// TwinCAT 3 PLC project EtherCAT_Test_1
// ProgramVersion: 3.1.4023.0
// libraries:
//   Tc2_EtherCAT, * (Beckhoff Automation GmbH)
//   Tc2_HVAC, * (Beckhoff Automation GmbH)
//   Tc2_Standard, * (Beckhoff Automation GmbH)
//   Tc2_System, * (Beckhoff Automation GmbH)
//   Tc3_Module, * (Beckhoff Automation GmbH)
// project tree:
//   DUTs/ ST_TypeOfPositioning.TcDUT
//   GVLs/ GVL.TcGVL
//   / PlcTask.TcTTO
//   POUs/ MAIN.TcPOU, P_ProfilePositionModeTest.TcPOU, StartUpTests.TcPOU, ST_PlcErrorStartUp.TcDUT
//   POUs/ProfilePositionMode/ FB_EnableDevice.TcPOU, Motion.TcPOU
// real-time tasks:
//   TASK PlcTask: cycle T#10ms, priority 20, ADS port 350
// motion (NC):
//   TASK NC-Task 1 SAF: cycle T#2ms, priority 4, ADS port 501
//   TASK NC-Task 1 SVB: cycle T#10ms, priority 8, ADS port 511
//   AXIS Axis 1 (id 1)
//     OtherSettings: AllowMotionCmdToSlave=true
//     encoder EncType=19
//       EncPara: MaxCount=#xffffffff
//     drive DrvType=16
//       DrvPara: MaxCount=#xffffffff
//         Analog: TorqueSetpointScale=10, ScaleFactorActTorque=0.1
//         TimeComp: TaskDelayCycles=1
//     controller CtrType=1
//       CtrPara: PriorControlFactor=1
//         Observer: BandWidth=20
// I/O:
//   DEVICE Device 1 (EtherCAT), AmsNetId 5.109.65.175.2.1
//     Term 1 (EK1200) [EK1200-5000 EtherCAT Power supply (2A E-Bus)]
//       Term 2 (EL1859) [EL1859 8Ch. Dig. Input 24V, 3ms, 8Ch. Dig. Output 24V, 0.5A]
//       Term 3 (EL6751) [EL6751 CANopen Master]
//       Term 4 (EK1110) [EK1110 EtherCAT extension]
//     Drive 5 (HTB) [HTB]
//       modules: Module 1 (csp - axis)

CONFIGURATION EtherCAT_Test_1
    RESOURCE PLC ON TwinCAT3
        TASK PlcTask(INTERVAL := T#10ms, PRIORITY := 20);
        PROGRAM MAIN WITH PlcTask : MAIN;
    END_RESOURCE
END_CONFIGURATION

// ---- DUTs/ST_TypeOfPositioning.TcDUT
TYPE ST_TypeOfPositioning :
STRUCT
	bStartImmediately			: BOOL; (*if Bool is true, target position is absolute, otherwise relative*)
	bAbsolutePositioning		: BOOL; (*if Bool is true, velocity does not change, when first target position is reached - no braking*)
	bChangeOnSetPoint			: BOOL; (*if set true, moving command is executed immediately*)
	nReferencing				: BYTE;
	(*describes positioning behaviour 
		- 1: Positioning relative to previous target position
		- 2: Positioning relative to default value of ramp generator
		- 3: Positioning relative to actual position*)	
END_STRUCT
END_TYPE

// ---- POUs/ST_PlcErrorStartUp.TcDUT
TYPE ST_PlcErrorStartUp :
STRUCT
	bPlcError		: BOOL;
	bErrorCode		: ARRAY[1..4] OF UDINT;
END_STRUCT
END_TYPE

// ---- GVLs/GVL.TcGVL
{attribute 'qualified_only'}
VAR_GLOBAL
	sNetId				: T_AmsNetId := '5.109.65.175.2.1';
	nSlaveAddr			: UINT := 1004;
	
	Controlword AT%Q*		: UINT;	
	Statusword AT%I*		: UINT;
END_VAR

// ---- POUs/MAIN.TcPOU
PROGRAM MAIN
VAR_INPUT
	Controlword AT%Q*		: UINT;	
	TargetPosition AT%Q*	: DINT;
END_VAR
VAR_OUTPUT
	Statusword AT%I*		: UINT;
END_VAR
VAR
	bStartUpTest			: BOOL;
END_VAR	

VAR
	aTemperatureObjects		: ARRAY[1..2] OF INT := [1,1]; 	//0x2200, 0x2202
	aMOPObjects				: ARRAY[1..2] OF INT := [1,1]; 	//0x6060, 0x6061
	aControlStatusWords		: ARRAY[1..2] OF INT := [1,1]; 	//0x6040, 0x6041
	bTargetPosition			: BOOL;							//0x607A
	
	fbSetToPPMode			: FB_EcCoeSdoWrite;
	bSetToPPMode			: BOOL;
	tSetToPPMode			: TON;
	nModeOfOperation		: UDINT := 1;
END_VAR

//StartUpTests(bTrigger := bStartUpTest,
//	aTemperatureObjects := aTemperatureObjects,
//	aControlStatusWords := aControlStatusWords,
//	aMOPObjects := aMOPObjects,
//	sNetID := GVL.sNetId,
//	nSlaveAddr := GVL.nSlaveAddr);

fbSetToPPMode(sNetId := GVL.sNetId, 
				nSlaveAddr := GVL.nSlaveAddr,
				nIndex := 16#6060,
				pSrcBuf := ADR(nModeOfOperation),
				cbBufLen := SIZEOF (nModeOfOperation),
				bExecute := bSetToPPMode);
tSetToPPMode(IN := bSetToPPMode,
				PT := T#250MS);
bSetToPPMode := TRUE;
IF tSetToPPMode.Q THEN
	P_ProfilePositionModeTest();	
END_IF

				



//Hallo Julian

END_PROGRAM

// ---- POUs/P_ProfilePositionModeTest.TcPOU
PROGRAM P_ProfilePositionModeTest
VAR
	fbMoveInProfilePosition			: Motion;
	fbGetCurrentPosition			: FB_EcCoeSdoRead;
	fbGetStatusword					: FB_EcCoeSdoRead;
	fbGetPositionWindow				: FB_EcCoeSdoRead;
	fbGetPositionDemandValue		: FB_EcCoeSdoRead;
	tWaitForCurrentPosition			: TON;
	tWaitForPositionDemandValue		: TON;
	tGetStatusword					: TON;
	bGetCurrentPosition				: BOOL;
	bMove							: BOOL; 
	bExecuteTimer					: BOOL;
	bGetStatusword					: BOOL;
	bGetParameters					: BOOL;
	bSetPositioningOptionCode		: BOOL;
	bGetPositionDemandValue			: BOOL;
	bBasicOperationAbsStarted		: BOOL;
	bBasicOperationAbsFinished		: BOOL := FALSE;
	bPositioningOptionCodeSet		: BOOL;
	bTargetReached					: BOOL;
	bTestAbsolutePositioning		: BOOL;
	nTargetPosition					: DINT;
	nCurrentPosition				: DINT;
	nTargetPositionBuf				: DINT;
	nPositionDemandValue			: DINT;
	nStatusword						: UINT;
	nPositionWindow					: UDINT;
	
	
	bTest							: BOOL;
	bAusprobieren					: BOOL;
END_VAR

VAR
	bBasicOperationAbs				: BOOL;
	bBasicOperationRel				: BOOL;
	bPositioningOptionCode			: BOOL;
END_VAR

//For Test Set of Setpoints
VAR
	bSetOfSetpointFinished 			: BOOL;
	nCurrentPositionBuf				: DINT;
	bSetPointSet					: BOOL;  //For both
	bSetOfSetpoints					: BOOL;
	bStartBasicOperationAbs			: BOOL;
	bTestSetOfSetpoints				: BOOL;
	bSetOfSetpointsFinished			: BOOL;
END_VAR

//Fo Test Change Immediately
VAR
	bTestChangeImmediately			: BOOL;
	bChangeImmediatelyFinished		: BOOL;
	bChangeImmediately				: BOOL;
END_VAR

//For test of relative Positioninig
VAR
	tSetPositioningOptionCode		: TON;
	fbSetPositioningOptionCode		: FB_EcCoeSdoWrite;
	bTestRelativePositioning		: BOOL;
	bRelativePositioningFinished	: BOOL;
	nPositioningOptionCode			: DINT;
	nCounter						: DINT;
END_VAR

tWaitForCurrentPosition(IN := bGetCurrentPosition,
							PT := T#10MS);
tGetStatusword(IN := bGetStatusword,
					PT := T#500MS);	
tSetPositioningOptionCode(IN := bSetPositioningOptionCode,
							PT := T#125MS);		
tWaitForPositionDemandValue(IN := bGetPositionDemandValue,
							PT := T#125MS);
IF tWaitForCurrentPosition.Q THEN
	bGetCurrentPosition := FALSE;
ELSE
	bGetCurrentPosition := TRUE;		
END_IF
fbMoveInProfilePosition(sNetID := GVL.sNetId,
						nSlaveAddr := GVL.nSlaveAddr,
						nTargetPosition := nTargetPosition,
						bMove := bMove);
fbGetStatusword(sNetId := GVL.sNetId,
				nSlaveAddr := GVL.nSlaveAddr,
				nIndex := 16#6041,
				nSubindex := 0,
				pDstBuf := ADR(nStatusWord),
				cbBufLen := SIZEOF(nStatusWord),
				bExecute := bGetStatusword);
fbGetCurrentPosition(sNetId := GVL.sNetId,
						nSlaveAddr := GVL.nSlaveAddr,
						nIndex := 16#6064,
						nSubIndex := 0,
						pDstBuf := ADR(nCurrentPosition),
						cbBufLen := SIZEOF(nCurrentPosition),
						bExecute := bGetCurrentPosition);
fbGetPositionWindow(sNetId := GVL.sNetId,
					nSlaveAddr := GVL.nSlaveAddr,
					nIndex := 16#6067,
					nSubIndex := 0,
					pDstBuf := ADR(nPositionWindow),
					cbBufLen := SIZEOF(nPositionWindow),
					bExecute := bGetParameters);
fbGetPositionDemandValue(sNetId := GVL.sNetId,
							nSlaveAddr := GVL.nSlaveAddr,
							nIndex := 16#60FC,
							nSubIndex := 0,
							pDstBuf := ADR(nPositionDemandValue),
							cbBufLen := SIZEOF(nPositionDemandValue),
							bExecute := bGetPositionDemandValue);
fbSetPositioningOptionCode(sNetId := GVL.sNetId,
							nSlaveAddr := GVL.nSlaveAddr,
							nIndex := 16#60F2,
							nSubindex := 0,
							pSrcBuf := ADR(nPositioningOptionCode),
							cbBufLen := SIZEOF(nPositioningOptionCode),
							bExecute := bSetPositioningOptionCode);
bGetParameters := TRUE;

IF bStartBasicOperationAbs THEN					
	//Basic Operation
	//Set-point is applied to the device
	//Move to absolute position is tested
	//Wait until Target reach Bit is set
	//Control if position is within error window
	
	//Target shall be an absolute value
	MAIN.Controlword.6 := 0;

	//Operation has not yet started and we are sure that initial position is obtained
	IF NOT bBasicOperationAbsStarted THEN
		nTargetPosition := nCurrentPosition + 5000000;
		//Start absolute positioning
		bMove := TRUE;	
		bBasicOperationAbsStarted := TRUE;
	END_IF
					
	//Target reached?
	bGetStatusword := TRUE;
	IF tGetStatusword.Q THEN
		IF NOT nStatusword.10 THEN
			bGetStatusword := FALSE;
		ELSIF ((nCurrentPosition >= nTargetPosition - nPositionWindow)
				AND (nCurrentPosition <= nTargetPosition + nPositionWindow)) 
				AND fbMoveInProfilePosition.bStartPositioning THEN
			//absolute Positionining
			bBasicOperationAbs := TRUE;
			bBasicOperationAbsFinished := TRUE;
			bStartBasicOperationAbs := FALSE;
		ELSIF fbMoveInProfilePosition.bStartPositioning THEN
			bBasicOperationAbs := FALSE;
			bBasicOperationAbsFinished := TRUE;
			bStartBasicOperationAbs := FALSE;
		END_IF
		bGetStatusword := FALSE;
	END_IF
END_IF

//Test SetOfSetpoints
IF bTestSetOfSetpoints AND bBasicOperationAbsFinished AND NOT bSetOfSetpointsFinished THEN
	IF NOT bSetPointSet THEN
		MAIN.Controlword.5 := 0;
		nTargetPosition := nCurrentPosition + 100000000;
		nTargetPositionBuf := nTargetPosition;
		nCurrentPositionBuf := nCurrentPosition + 10000000/2;
		bSetPointSet := TRUE;
	END_IF
	IF (nCurrentPosition > nCurrentPositionBuf) AND bSetPointSet THEN
		nTargetPosition := nCurrentPositionBuf - 10000000/2;
	END_IF
	bSetOfSetpoints := TestChangeOfSetpoints(bActive => bSetOfSetpointsFinished);
	IF bSetOfSetpointsFinished THEN
		bSetPointSet := FALSE;
	END_IF
END_IF

//Change Immediately
IF bTestChangeImmediately AND bSetOfSetpointsFinished AND NOT bChangeImmediatelyFinished THEN
	IF NOT bSetPointSet THEN
		MAIN.Controlword.5 := 1;
		nTargetPosition := nCurrentPosition + 100000000;
		nTargetPositionBuf := nTargetPosition;
		nCurrentPositionBuf := nCurrentPosition + 10000000/2;
		bSetPointSet := TRUE;
	END_IF
	IF (nCurrentPosition > nCurrentPositionBuf) AND bSetPointSet THEN
		nTargetPosition := nCurrentPositionBuf - 10000000/2;
	END_IF
	bChangeImmediately := NOT TestChangeOfSetpoints(bActive => bChangeImmediatelyFinished);
END_IF

//Test relative positioning:
//Bit 6 of Controlword is set to 1

IF bTestRelativePositioning THEN
	MAIN.Controlword.6 := 1;
	//positioning option code: 0
	//Positioning moves shall be performed relative to the preciding
	//target position
	IF nCounter = 0 THEN
		nPositioningOptionCode := 0;
		IF tSetPositioningOptionCode.Q THEN
			nTargetPosition := 5000000;
		END_IF
		
		nCounter := nCounter + 1;
	END_IF

	//positioning option code: 2#0001
	//Positioning moves shall be performed relative to the actual
	//positioning demand value (16#60FC)
	
	//positioning option code : 2#0010
	//Positioning moves shall be performed relative to the position
	//actual value (16#6064)
END_IF

//test

METHOD TestChangeOfSetpoints : BOOL
VAR_OUTPUT
	bActive		: BOOL;
END_VAR
IF ((nCurrentPosition >= nTargetPositionBuf - nPositionWindow)
	AND (nCurrentPosition <= nTargetPositionBuf + nPositionWindow)) THEN
	bActive := TRUE;
	bSetOfSetPointsFinished := TRUE;
ELSIF ((nCurrentPosition >= nTargetPosition - nPositionWindow)
	AND (nCurrentPosition <= nTargetPosition + nPositionWindow)) THEN
	TestChangeOfSetpoints := FALSE;
	bActive := TRUE;
END_IF
END_METHOD

END_PROGRAM

// ---- POUs/ProfilePositionMode/Motion.TcPOU
FUNCTION_BLOCK Motion
VAR_INPUT
	sNetID					: T_AmsNetId;
	nSlaveAddr				: UINT;
	nTargetPosition			: DINT;
END_VAR
VAR_OUTPUT
	bSuccess				: BOOL;
	bSetpointSet			: BOOL;
	bStartPositioning		: BOOL;
END_VAR
VAR_IN_OUT
//	aControlStatusWords		: ARRAY[1..2] OF INT; 			//0x6040 (Controlword), 0x6041 (Statusword)  
//	bTargetPosition			: BOOL;							//0x607A (Target Position)
	bMove					: BOOL;
END_VAR
VAR
	eMotionState			: (WAIT_FOR_TRIGGER, ENABLE_DEVICE, SET_SETPOINT, VALIDATE_SETPOINT, ACKNOWLEDGE_SET_POINT, WAIT_FOR_NEW_SETPOINT);
	fbEnableDevice			: FB_EnableDevice;
	fbSetSetpoint			: FB_EcCoeSdoWrite;
	fbGetStatusword			: FB_EcCoeSdoRead;
	tWait					: TON;
	tWait2					: TON;
	rTrig					: R_TRIG;
	nStatusword				: UINT;
	bGetStatusword			: BOOL;
	bExecuteWait			: BOOL;
	bSetSetpoint			: BOOL;
	nSetPointBuf			: DINT;
END_VAR

CASE eMotionState OF
	WAIT_FOR_TRIGGER:
		MAIN.Controlword := 0;
		bStartPositioning := FALSE;
		IF bMove THEN
			bSetpointSet := TRUE;
			bSuccess := TRUE;
			ADSLOGSTR(msgCtrlMask := ADSLOG_MSGTYPE_HINT,
				msgFmtStr := 'Enable Device',
				strArg := '');
			eMotionState := ENABLE_DEVICE;
		END_IF	

	ENABLE_DEVICE:
		fbEnableDevice (bTrigger := bMove,
						bSuccess => bSuccess,
						sNetId := sNetId,
						nSlaveAddr := nSlaveAddr);
		IF fbEnableDevice.bFinished THEN
			IF NOT bSuccess THEN
//				aControlStatusWords[1] := 0;
//				aControlStatusWords[2] := 0;
				ADSLOGSTR(msgCtrlMask := ADSLOG_MSGTYPE_HINT,
					msgFmtStr := 'Device not successfully enabled',
					strArg := '');
				eMotionState := WAIT_FOR_TRIGGER;
			ELSE
				ADSLOGSTR(msgCtrlMask := ADSLOG_MSGTYPE_HINT,
					msgFmtStr := 'Device successfully enabled',
					strArg := '');
				eMotionState := SET_SETPOINT;
			END_IF
		END_IF
		
	WAIT_FOR_NEW_SETPOINT:
		IF nTargetPosition <> nSetPointBuf THEN
			ADSLOGSTR(msgCtrlMask := ADSLOG_MSGTYPE_HINT,
				msgFmtStr := 'Set Setpoint',
				strArg := '');
				bStartPositioning := FALSE;
			eMotionState := SET_SETPOINT;
		END_IF
		
	SET_SETPOINT:
		bSetpointSet	:= TRUE;
		nSetPointBuf := nTargetPosition;
		fbSetSetpoint(sNetId := sNetID,
					nSlaveAddr := nSlaveAddr,
					nSubIndex := 0,
					nIndex := 16#607A,
					pSrcBuf := ADR(nTargetPosition),
					cbBufLen := SIZEOF(nTargetPosition),
					bExecute := bSetSetpoint);
		bSetSetpoint := TRUE;
		MAIN.TargetPosition := nTargetPosition;
		tWait(IN := bExecuteWait,
				PT := T#175MS); 
		bExecuteWait := TRUE;
		IF tWait.Q THEN
			bExecuteWait := FALSE;
			IF fbSetSetpoint.bError THEN
				//Error when setting Target Position
				bSuccess := FALSE;
				bSetSetpoint := FALSE;
				eMotionState := WAIT_FOR_TRIGGER;
			ELSE
				ADSLOGSTR(msgCtrlMask := ADSLOG_MSGTYPE_HINT,
					msgFmtStr := 'Validate Setpoint',
					strArg := '');
				eMotionState := VALIDATE_SETPOINT;
			END_IF
		END_IF
 
	VALIDATE_SETPOINT:
		bExecuteWait := TRUE;
		MAIN.Controlword.4 := 1;
		fbGetStatusword(sNetId := sNetId,
			nSlaveAddr := nSlaveAddr,
			nIndex := 16#6041,
			nSubIndex := 0,
			pDstBuf := ADR(nStatusword),
			cbBufLen := SIZEOF(nStatusword),
			bExecute := bGetStatusword);
		IF tWait.Q THEN
			bExecuteWait := FALSE;
			tWait2(IN := bGetStatusword,
				PT := T#250MS);
			bGetStatusword := TRUE;
			IF tWait2.Q THEN
				bGetStatusword := FALSE;
				IF nStatusword.12 THEN
					eMotionState := ACKNOWLEDGE_SET_POINT;
				ELSE 
					bSetSetpoint := FALSE;
					bSuccess := FALSE;
//					aControlStatusWords[1] := 0;
//					aControlStatusWords[2] := 0;
					ADSLOGSTR(msgCtrlMask := ADSLOG_MSGTYPE_HINT,
						msgFmtStr := 'Error when validating setpoint',
						strArg := '');
					eMotionState := WAIT_FOR_TRIGGER;
				END_IF
			END_IF
		END_IF
		
	ACKNOWLEDGE_SET_POINT:
		ADSLOGSTR(msgCtrlMask := ADSLOG_MSGTYPE_HINT,
			msgFmtStr := 'Acknowledge Setpoint',
			strArg := '');
		bGetStatusword := TRUE;
		IF tWait2.Q AND nStatusword.12 THEN
			bStartPositioning := TRUE;
			bGetStatusword := FALSE;
			//Set point acknowledge is set back
			MAIN.Controlword.4 := 0;
			ADSLOGSTR(msgCtrlMask := ADSLOG_MSGTYPE_HINT,
				msgFmtStr := 'Wait for new Setpoint',
				strArg := '');
			eMotionState := WAIT_FOR_NEW_SETPOINT;
		ELSE
			//TODO FAULT
			eMotionState := WAIT_FOR_TRIGGER;
		END_IF
END_CASE

END_FUNCTION_BLOCK

// ---- POUs/ProfilePositionMode/FB_EnableDevice.TcPOU
FUNCTION_BLOCK FB_EnableDevice 
VAR_IN_OUT
	bTrigger			: BOOL;
END_VAR
VAR_INPUT
	sNetID				: T_AmsNetId;
	nSlaveAddr			: UINT;
END_VAR
VAR_OUTPUT
	bFinished			: BOOL;
	bSuccess			: BOOL;
END_VAR
VAR
	eState				: (WAIT_FOR_TRIGGER, SHUTDOWN, SWITCH_ON);
	tWait1				: TON;
	tWait2				: TON;
	fbGetStatusword		: FB_EcCoeSdoRead;
	nStatusword			: UINT;
	bGetStatusword		: BOOL;
	bExecuteTimer		: BOOL;
END_VAR

CASE eState OF
	WAIT_FOR_TRIGGER:
		IF bTrigger THEN
			bExecuteTimer	:= FALSE;
			bSuccess := TRUE;
			bFinished := FALSE;
			bTrigger := FALSE;
			eState := SHUTDOWN;
		END_IF
	
	SHUTDOWN:
		MAIN.Controlword.0 := 0;
		MAIN.Controlword.1 := 1;
		MAIN.Controlword.2 := 1;
		MAIN.Controlword.7 := 0;

		tWait1(PT := T#125MS,
			IN := bExecuteTimer);
			bExecuteTimer := TRUE;
		IF tWait1.Q THEN
			bExecuteTimer := FALSE;
			tWait2(IN := bGetStatusword,
				PT := T#250MS);
			fbGetStatusword(sNetId := sNetId,
				nSlaveAddr := nSlaveAddr,
				nIndex := 16#6041,
				nSubIndex := 0,
				pDstBuf := ADR(nStatusword),
				cbBufLen := SIZEOF(nStatusword),
				bExecute := bGetStatusword);
			bGetStatusword := TRUE;
			IF tWait2.Q THEN
				ADSLOGSTR(msgCtrlMask := ADSLOG_MSGTYPE_HINT,
					msgFmtStr := 'Shutdown',
					strArg := '');
				bExecuteTimer := FALSE;
				IF (nStatusword.0 = 1 AND nStatusword.5) 
					AND NOT (nStatusword.1 AND nStatusword.2 AND nStatusword.3
						AND nStatusword.6) THEN
 					eState := SWITCH_ON;
				ELSE 
					bSuccess := FALSE;
					bFinished := TRUE;
					eState := WAIT_FOR_TRIGGER;
				END_IF
			END_IF
		END_IF
		
	SWITCH_ON:
		ADSLOGSTR(msgCtrlMask := ADSLOG_MSGTYPE_HINT,
			msgFmtStr := 'Switch On',
			strArg := '');
		MAIN.Controlword.0 := 1;
		MAIN.Controlword.1 := 1;
		MAIN.Controlword.2 := 1;
		Main.Controlword.3 := 1;
		Main.Controlword.7 := 0;
		bExecuteTimer := TRUE;
		bGetStatusWord := TRUE;
		IF tWait1.Q THEN
			bExecuteTimer	:= FALSE;
			IF tWait2.Q THEN
				bGetStatusword := FALSE;
				IF nStatusword.0 AND nStatusword.1 AND nStatusword.5 
						AND NOT (nStatusword.2 AND nStatusword.3 AND nStatusword.6) THEN
					bSuccess := FALSE;
				END_IF
				bFinished := TRUE;
				eState := WAIT_FOR_TRIGGER;
			END_IF
		END_IF
END_CASE

END_FUNCTION_BLOCK

// ---- POUs/StartUpTests.TcPOU
PROGRAM StartUpTests
VAR CONSTANT
	stPlcErrorInit			: ST_PlcErrorStartUp := (bPlcError := FALSE, bErrorCode := [0,0,0,0]);
END_VAR

VAR
	eStartUpState 			: (WAIT_FOR_TRIGGER, TEST_SWITCH_ON_DISABLED, 
								SET_MODE_OF_OPERATION, TEST_MODE_OF_OPERATION, GET_TEMPERATURE, CHECK_PLC_ERROR);
	fbSetModeOfOperation	: FB_EcCoeSdoWrite;
	fbGetModeOfOperation	: FB_EcCoeSdoRead;
	fbGetDriveTemperature	: FB_EcCoeSdoRead;
	fbGetMotorTemperature	: FB_EcCoeSdoRead;
	stPlcError				: ST_PlcErrorStartUp;
	tTimeout				: TON;
	tWait1					: TON;
	tWait2					: TON;
	tWait					: TON;
	counter					: INT := -1;
	modeOfOperation			: INT;
	bExecuteChangeMOP		: BOOL;	
	bTestChangeMOP			: BOOL;
END_VAR
VAR_IN_OUT
	bTrigger				: BOOL;
	aTemperatureObjects		: ARRAY[1..2] OF INT;
	aMOPObjects				: ARRAY[1..2] OF INT;
	aControlStatusWords		: ARRAY[1..2] OF INT;
END_VAR
VAR_OUTPUT
	bSwitchOnDisabled		: BOOL;
	bChangeModeOfOperation	: BOOL := TRUE;
	bFinished				: BOOL;
	nDriveTemperature		: INT;
	nMotorTemperature		: INT;
END_VAR
VAR_INPUT
	sNetID					: T_AmsNetId;
	nSlaveAddr				: UINT;
END_VAR

CASE eStartUpState OF
	WAIT_FOR_TRIGGER:
		IF bTrigger THEN
			bTrigger := FALSE;
			tTimeout.IN := FALSE;
			bSwitchOnDisabled := FALSE;
			bChangeModeOfOperation := FALSE;
			bFinished := FALSE;
			counter := 1;
			stPlcError := stPlcErrorInit;
			eStartUpState := TEST_SWITCH_ON_DISABLED;
		END_IF
	
	TEST_SWITCH_ON_DISABLED:
		tTimeout(IN := TRUE,
			PT := T#1000MS);
		IF MAIN.Statusword.6 THEN
			bSwitchOnDisabled := TRUE;
			eStartUpState := SET_MODE_OF_OPERATION;
		ELSIF tTimeout.Q THEN
			bSwitchOnDisabled := FALSE;
			aControlStatusWords[1] := 0;
			eStartUpState := SET_MODE_OF_OPERATION;
		END_IF
	
	SET_MODE_OF_OPERATION:
	bTestChangeMOP := FALSE;
		fbSetModeOfOperation(sNetId := sNetId,
							nSlaveAddr := nSlaveAddr,
							nSubIndex := 0,
							nIndex := 16#6060,
							pSrcBuf := ADR(counter),
							cbBufLen := SIZEOF(counter),
							bExecute := bExecuteChangeMOP);
		tWait1(PT := T#2S, 
			IN := bExecuteChangeMOP);
		bExecuteChangeMOP := TRUE;				
		IF tWait1.Q THEN
			eStartUpState := TEST_MODE_OF_OPERATION;
		END_IF

	TEST_MODE_OF_OPERATION:
		bExecuteChangeMOP := FALSE;	
		fbGetModeOfOperation(sNetId := sNetId,
							nSlaveAddr := nSlaveAddr,
							nSubIndex := 0,
							nIndex := 16#6061,
							pDstBuf := ADR(modeOfOperation),
							cbBufLen := SIZEOF(modeOfOperation),
							bExecute := bTestChangeMOP);
		tWait2(PT := T#2S,
				IN := bTestChangeMOP);
		bTestChangeMOP := TRUE; 
		IF tWait2.Q THEN
			IF NOT modeOfOperation = counter AND counter <> 5 THEN
				bChangeModeOfOperation := FALSE;
				aMOPObjects[1] := 0;
				aMOPObjects[2] := 0;
			END_IF
			counter := counter + 1;
			IF counter < 11 THEN
				eStartUpState := SET_MODE_OF_OPERATION;
			ELSE
				eStartUpState := GET_TEMPERATURE;
			END_IF
		END_IF
	
	GET_TEMPERATURE:
		fbGetDriveTemperature(sNetId := sNetId,
							nSlaveAddr := nSlaveAddr,
							nSubIndex := 0,
							nIndex := 16#2200,
							pDstBuf := ADR(nDriveTemperature),
							cbBufLen := SIZEOF(nDriveTemperature),
							bExecute := TRUE);
		fbGetMotorTemperature(sNetId := sNetId,
							nSlaveAddr := nSlaveAddr,
							nSubIndex := 0,
							nIndex := 16#2202,
							pDstBuf := ADR(nMotorTemperature),
							bExecute := TRUE);							
		tWait(IN := TRUE,
			PT := T#125MS);
		IF tWait.Q THEN
			tWait.IN := FALSE;
		//	eStartUpState := CHECK_PLC_ERROR;
		END_IF
		
		CHECK_PLC_ERROR:
			IF fbSetModeOfOperation.bError OR fbGetModeOfOperation.bError OR
				fbGetDriveTemperature.bError OR fbGetMotorTemperature.bError THEN
				stPlcError.bPlcError := TRUE;
				IF fbSetModeOfOperation.bError THEN
					stPlcError.bErrorCode[1] := fbSetModeOfOperation.nErrId;
					aMOPObjects[1] := 0;
				END_IF
				IF fbGetModeOfOperation.bError THEN
					stPlcError.bErrorCode[2] := fbGetModeOfOperation.nErrId;
					aMOPObjects[2] := 0;		
				END_IF
				IF fbGetDriveTemperature.bError THEN
					stPlcError.bErrorCode[3] := fbGetDriveTemperature.nErrId;
					aTemperatureObjects[1] := 0;
				END_IF
				IF fbGetMotorTemperature.bError THEN
					stPlcError.bErrorCode[4] := fbGetMotorTemperature.nErrId;
					aTemperatureObjects[2] := 0;
				END_IF
			END_IF
			bFinished := TRUE;
			eStartUpState := WAIT_FOR_TRIGGER;
END_CASE

END_PROGRAM
